// TwinCAT 3 PLC project OEF_1
// ProgramVersion: 3.1.4024.0
// libraries:
//   Tc2_BABasic, * (Beckhoff Automation GmbH)
//   Tc2_Standard, * (Beckhoff Automation GmbH)
//   Tc2_System, * (Beckhoff Automation GmbH)
//   Tc3_Module, * (Beckhoff Automation GmbH)
// project tree:
//   / GlobalTextList.TcGTLO, PlcTask.TcTTO, Visualization Manager.TcVMO (not stored)
//   POUs/ MAIN.TcPOU
//   VISUs/ Visualization.TcVIS

CONFIGURATION OEF_1
    RESOURCE PLC ON TwinCAT3
        TASK PlcTask(INTERVAL := T#10ms, PRIORITY := 20);
        PROGRAM MAIN WITH PlcTask : MAIN;
    END_RESOURCE
END_CONFIGURATION

// ---- POUs/MAIN.TcPOU
PROGRAM MAIN
VAR
	bLed1 AT %Q*: BOOL := FALSE;
	
	BButton1 AT %I*: BOOL := false;
	bButton2 AT %I*: BOOL := FALSE;
	bButton3 AT %I*: BOOL := FALSE;
	
	bTriggerLong: BOOL;
	bTriggerShort: BOOL;
	
	FB_Timer_Setting: CTUD ;
	fbtimer: TON;
	FB_Button: FB_ShortLongClick;
	FB_Lights: FB_Light;
	fbWarning: TOF;
	fbBlinking: TOF;
	fbTON: TON := (PT := TIME#500MS);
	bLED2 AT %Q*: BOOL;
END_VAR

FB_Button(bSwitch:= BButton1, tSwitchTime:= T#2S, bShortClick=> bTriggerShort , bLongClick=> bTriggerLong);
FB_Lights(bOn:=  , bOff:= fbtimer.q, bToggle:= bTriggerShort, bLight=>bLed1 );
FB_Timer_Setting(CU:= bButton2, CD:= bButton3 );
fbtimer(IN:= bLed1 AND NOT bTriggerLong , PT:=  TO_TIME(FB_Timer_Setting.CV * 1000 + 3*1000));
fbBlinking(IN:= fbTimer.ET = TO_TIME(fb_timer_setting.CV * 1000), PT:= T#3S);
IF fbBlinking.Q THEN
	fbTON(IN:= NOT(fbTON.Q), Q=>bLED2);
END_IF

END_PROGRAM

// ---- VISUs/Visualization.TcVIS
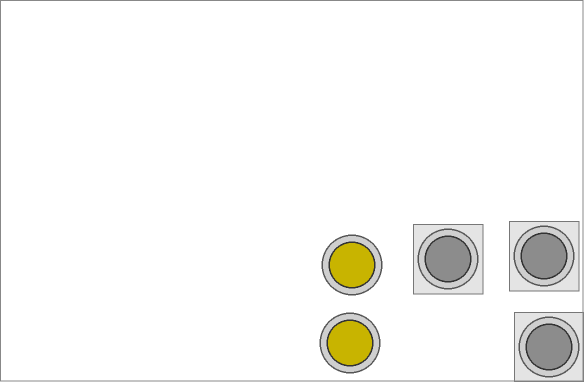
VISUALIZATION Visualization  // 584x382
    Lamp1 (317,230 70x70), variable: MAIN.bLed1, style: Lamp-Lamp1-Yellow
    Lamp1 (315,308 70x70), variable: MAIN.bLED2, style: Lamp-Lamp1-Yellow
    PushSwitch (413,224 70x70), variable: MAIN.BButton1, behaviour: TAP, style: Switch-PushSwitch-Gray
    PushSwitch (509,221 70x70), variable: MAIN.bButton2, behaviour: TAP, style: Switch-PushSwitch-Gray
    PushSwitch (514,312 70x70), variable: MAIN.bButton3, behaviour: TAP, style: Switch-PushSwitch-Gray
END_VISUALIZATION
